TYPE Terminal_Output_typ : 	
	STRUCT  
		Status:  Terminal_Status_typ;
		Monitor: Terminal_Monitor_typ;
	END_STRUCT
END_TYPE

(* stored: Version 1.1.0.1, ProductVersion 3.1.4024.3
   DUT Terminal_Output_typ: Id {6b63e8c1-3140-0659-2aa8-b2e3c03818a5} *)
